// TIA Portal V19 export
TYPE "lexchangetray_typeUnEmn_interface"
// Type: lexchangetray_typeUnEmn_recieve_interface
// Type: lexchangetray_typeUnEmn_deliver_interface
// stored: Access Published
   STRUCT
      deliver : "lexchangetray_typeUnEmn_deliver_interface";
      recieve : "lexchangetray_typeUnEmn_recieve_interface";
   END_STRUCT;
END_TYPE
